DATA_BLOCK "照明通风_DB"
{ S7_Optimized_Access := 'TRUE' }
VERSION : 0.1
NON_RETAIN
"照明通风"

BEGIN

END_DATA_BLOCK

